TYPE "TMeasuring_STATUSWORD"
VERSION : 0.1
// Block: TMeasuring_STATUSWORD
   STRUCT
      Control : Bool;
      Error : Bool;
      RestartActive : Bool;
      OnlineStartValuesChanged : Bool;
      CommunicationOK : Bool;
   END_STRUCT;

END_TYPE
